ABB RAPID module: 0056609E

MODULE SERVER

!////////////////
!GLOBAL VARIABLES
!////////////////

!//Robot configuration
PERS tooldata currentTool := [TRUE,[[0,0,0],[1,0,0,0]],[0.001,[0,0,0.001],[1,0,0,0],0,0,0]];
PERS wobjdata currentWobj := [FALSE,TRUE,"",[[0,0,0],[1,0,0,0]],[[500,0,500],[0,0,1,0]]];
PERS speeddata currentSpeed;
PERS zonedata currentZone;
!//NOTE:To modify the default values go to the method Initialize

!//PC communication
VAR socketdev clientSocket;
VAR socketdev serverSocket;
VAR num instructionCode;
VAR num params{10};
VAR num nParams;
!PERS string ipController:= "192.168.180.128";
!PERS string ipController:= "127.0.0.1"; !localhost
PERS string ipController:= "192.168.1.7"; !mlab Network
PERS num serverPort:= 5000;

!//Motion of the robot
VAR robtarget cartesianTarget;
VAR jointtarget jointsTarget;
VAR bool moveCompleted; !Set to true after finishing a Move instruction.

!//Correct Instruction Execution and possible return values
VAR num ok;
CONST num SERVER_BAD_MSG :=  0;
CONST num SERVER_OK := 1;




!////////////////
!LOCAL METHODS
!////////////////

!//Method to parse the message received from a PC
!// If correct message, loads values on:
!// - instructionCode.
!// - nParams: Number of received parameters.
!// - params{nParams}: Vector of received params.
PROC ParseMsg(string msg)
    !//Local variables
    VAR bool auxOk;
    VAR num ind:=1;
    VAR num newInd;
    VAR num length;
    VAR num indParam:=1;
    VAR string subString;
    VAR bool end := FALSE;

    !//Find the end character
    length := StrMatch(msg,1,"#");
    IF length > StrLen(msg) THEN
        !//Corrupt message
        nParams := -1;
    ELSE
        !//Read Instruction code
        newInd := StrMatch(msg,ind," ") + 1;
        subString := StrPart(msg,ind,newInd - ind - 1);
        auxOk:= StrToVal(subString, instructionCode);
        IF auxOk = FALSE THEN
            !//Impossible to read instruction code
            nParams := -1;
        ELSE
            ind := newInd;
            !//Read all instruction parameters (maximum of 8)
            WHILE end = FALSE DO
                newInd := StrMatch(msg,ind," ") + 1;
                IF newInd > length THEN
                    end := TRUE;
                ELSE
                    subString := StrPart(msg,ind,newInd - ind - 1);
                    auxOk := StrToVal(subString, params{indParam});
                    indParam := indParam + 1;
                    ind := newInd;
                ENDIF
            ENDWHILE
            nParams:= indParam - 1;
        ENDIF
    ENDIF
ENDPROC


!//Handshake between server and client:
!// - Creates socket.
!// - Waits for incoming TCP connection.
PROC ServerCreateAndConnect(string ip, num port)
    VAR string clientIP;

    SocketCreate serverSocket;
    SocketBind serverSocket, ip, port;
    SocketListen serverSocket;
    TPWrite "SERVER: Server waiting for incomming connections ...";
    WHILE SocketGetStatus(clientSocket) <> SOCKET_CONNECTED DO
        SocketAccept serverSocket,clientSocket \ClientAddress:=clientIP \Time:=WAIT_MAX;
        IF SocketGetStatus(clientSocket) <> SOCKET_CONNECTED THEN
            TPWrite "SERVER: Problem serving an incomming connection.";
            TPWrite "SERVER: Try reconnecting.";
        ENDIF
        !//Wait 0.5 seconds for the next reconnection
        WaitTime 0.5;
    ENDWHILE
    TPWrite "SERVER: Connected to IP " + clientIP;
ENDPROC


!//Parameter initialization
!// Loads default values for
!// - Tool.
!// - WorkObject.
!// - Zone.
!// - Speed.
PROC Initialize()
    currentTool := [TRUE,[[0,0,0],[1,0,0,0]],[0.001,[0,0,0.001],[1,0,0,0],0,0,0]];
    currentWobj := [FALSE,TRUE,"",[[0,0,0],[1,0,0,0]],[[0,0,0],[1,0,0,0]]];
    currentSpeed := [100, 50, 0, 0];
    currentZone := [FALSE, 0.3, 0.3,0.3,0.03,0.3,0.03]; !z0
ENDPROC


!////////////////////////
!//SERVER: Main procedure
!////////////////////////
PROC main()
    !//Local variables
    VAR string receivedString;   !//Received string
    VAR string sendString;       !//Reply string
    VAR string addString;        !//String to add to the reply.
    VAR bool connected;          !//Client connected
    VAR bool reconnected;        !//Drop and reconnection happened during serving a command
    VAR robtarget cartesianPose;
    VAR jointtarget jointsPose;

    !//Motion configuration
    ConfL \Off;
    SingArea \Wrist;
    moveCompleted:= TRUE;

    !//Initialization of WorkObject, Tool, Speed and Zone
    Initialize;

    !//Socket connection
    connected:=FALSE;
    ServerCreateAndConnect ipController,serverPort;
    connected:=TRUE;

    !//Server Loop
    WHILE TRUE DO
        !//Initialization of program flow variables
        ok:=SERVER_OK;              !//Correctness of executed instruction.
        reconnected:=FALSE;         !//Has communication dropped after receiving a command?
        addString := "";

        !//Wait for a command
        SocketReceive clientSocket \Str:=receivedString \Time:=WAIT_MAX;
        ParseMsg receivedString;

        !//Execution of the command
        TEST instructionCode
            CASE 0: !Ping
                IF nParams = 0 THEN
                    ok := SERVER_OK;
                ELSE
                    ok := SERVER_BAD_MSG;
                ENDIF
            CASE 1: !Cartesian Move
                IF nParams = 7 THEN
                    cartesianTarget :=[[params{1},params{2},params{3}],
                                       [params{4},params{5},params{6},params{7}],
                                       [0,0,0,0],
                                       [9E9,9E9,9E9,9E9,9E9,9E9]];
                    ok := SERVER_OK;
                    moveCompleted := FALSE;
                    MoveL cartesianTarget, currentSpeed, currentZone, currentTool \WObj:=currentWobj ;
                    moveCompleted := TRUE;
                ELSE
                    ok := SERVER_BAD_MSG;
                ENDIF
            CASE 2: !Joint Move
                IF nParams = 6 THEN
                    jointsTarget:=[[params{1},params{2},params{3},params{4},params{5},params{6}],
                                   [0, 9E9, 9E9, 9E9, 9E9, 9E9]];
                    ok := SERVER_OK;
                    moveCompleted := FALSE;
                    MoveAbsJ jointsTarget, currentSpeed, currentZone, currentTool \Wobj:=currentWobj;
                    moveCompleted := TRUE;
                ELSE
                    ok :=SERVER_BAD_MSG;
                ENDIF
            CASE 3: !Get Cartesian Coordinates (with current tool and workobject)
                IF nParams = 0 THEN
                    cartesianPose := CRobT(\Tool:=currentTool \WObj:=currentWObj);
                    addString := NumToStr(cartesianPose.trans.x,2) + " ";
                    addString := addString + NumToStr(cartesianPose.trans.y,2) + " ";
                    addString := addString + NumToStr(cartesianPose.trans.z,2) + " ";
                    addString := addString + NumToStr(cartesianPose.rot.q1,3) + " ";
                    addString := addString + NumToStr(cartesianPose.rot.q2,3) + " ";
                    addString := addString + NumToStr(cartesianPose.rot.q3,3) + " ";
                    addString := addString + NumToStr(cartesianPose.rot.q4,3); !End of string
                    ok := SERVER_OK;
                ELSE
                    ok :=SERVER_BAD_MSG;
                ENDIF
            CASE 4: !Get Joint Coordinates
                IF nParams = 0 THEN
                    jointsPose := CJointT();
                    addString := NumToStr(jointsPose.robax.rax_1,2) + " ";
                    addString := addString + NumToStr(jointsPose.robax.rax_2,2) + " ";
                    addString := addString + NumToStr(jointsPose.robax.rax_3,2) + " ";
                    addString := addString + NumToStr(jointsPose.robax.rax_4,2) + " ";
                    addString := addString + NumToStr(jointsPose.robax.rax_5,2) + " ";
                    addString := addString + NumToStr(jointsPose.robax.rax_6,2); !End of string
                    ok := SERVER_OK;
                ELSE
                    ok:=SERVER_BAD_MSG;
                ENDIF
            CASE 6: !Set Tool
                IF nParams = 7 THEN
                    currentTool.tframe.trans.x:=params{1};
                    currentTool.tframe.trans.y:=params{2};
                    currentTool.tframe.trans.z:=params{3};
                    currentTool.tframe.rot.q1:=params{4};
                    currentTool.tframe.rot.q2:=params{5};
                    currentTool.tframe.rot.q3:=params{6};
                    currentTool.tframe.rot.q4:=params{7};
                    ok := SERVER_OK;
                ELSE
                    ok:=SERVER_BAD_MSG;
                ENDIF
            CASE 7: !Specify Work Object
                IF nParams = 7 THEN
                    currentWobj.oframe.trans.x:=params{1};
                    currentWobj.oframe.trans.y:=params{2};
                    currentWobj.oframe.trans.z:=params{3};
                    currentWobj.oframe.rot.q1:=params{4};
                    currentWobj.oframe.rot.q2:=params{5};
                    currentWobj.oframe.rot.q3:=params{6};
                    currentWobj.oframe.rot.q4:=params{7};
                    ok := SERVER_OK;
                ELSE
                    ok:=SERVER_BAD_MSG;
                ENDIF
            CASE 8: !Specify Speed of the Robot
                IF nParams = 4 THEN
                    currentSpeed.v_tcp:=params{1};
                    currentSpeed.v_ori:=params{2};
                    currentSpeed.v_leax:=params{3};
                    currentSpeed.v_reax:=params{4};
                    ok := SERVER_OK;
                ELSE
                    ok:=SERVER_BAD_MSG;
                ENDIF
            CASE 9: !Specify ZoneData
                IF nParams = 4 THEN
                    IF params{1}=1 THEN
                        currentZone.finep := TRUE;
                        currentZone.pzone_tcp := 0.0;
                        currentZone.pzone_ori := 0.0;
                        currentZone.zone_ori := 0.0;
                    ELSE
                        currentZone.finep := FALSE;
                        currentZone.pzone_tcp := params{2};
                        currentZone.pzone_ori := params{3};
                        currentZone.zone_ori := params{4};
                    ENDIF
                    ok := SERVER_OK;
                ELSE
                    ok:=SERVER_BAD_MSG;
                ENDIF
            CASE 99: !Close Connection
                IF nParams = 0 THEN
                    TPWrite "SERVER: Client has closed connection.";
                    connected := FALSE;
                    !//Closing the server
                    SocketClose clientSocket;
                    SocketClose serverSocket;

                    !Reinitiate the server
                    ServerCreateAndConnect ipController,serverPort;
                    connected := TRUE;
                    reconnected := TRUE;
                    ok := SERVER_OK;
                ELSE
                    ok := SERVER_BAD_MSG;
                ENDIF
            DEFAULT:
                TPWrite "SERVER: Illegal instruction code";
                ok := SERVER_BAD_MSG;
        ENDTEST

        !Compose the acknowledge string to send back to the client
        IF connected = TRUE THEN
            IF reconnected = FALSE THEN
			    IF SocketGetStatus(clientSocket) = SOCKET_CONNECTED THEN
				    sendString := NumToStr(instructionCode,0);
                    sendString := sendString + " " + NumToStr(ok,0);
                    sendString := sendString + " " + addString;
                    SocketSend clientSocket \Str:=sendString;
			    ENDIF
            ENDIF
        ENDIF
    ENDWHILE

ERROR (LONG_JMP_ALL_ERR)
    TPWrite "SERVER: ------";
    TPWrite "SERVER: Error Handler:" + NumtoStr(ERRNO,0);
    TEST ERRNO
        CASE ERR_SOCK_CLOSED:
            TPWrite "SERVER: Lost connection to the client.";
            TPWrite "SERVER: Closing socket and restarting.";
            TPWrite "SERVER: ------";
            connected:=FALSE;
            !//Closing the server
            SocketClose clientSocket;
            SocketClose serverSocket;
            !//Reinitiate the server
            ServerCreateAndConnect ipController,serverPort;
            reconnected:= TRUE;
            connected:= TRUE;
            RETRY;
        DEFAULT:
            TPWrite "SERVER: Unknown error.";
            TPWrite "SERVER: Closing socket and restarting.";
            TPWrite "SERVER: ------";
            connected:=FALSE;
            !//Closing the server
            SocketClose clientSocket;
            SocketClose serverSocket;
            !//Reinitiate the server
            ServerCreateAndConnect ipController,serverPort;
            reconnected:= TRUE;
            connected:= TRUE;
            RETRY;
    ENDTEST
ENDPROC

ENDMODULE
